{attribute 'linkalways'} 
{attribute 'no_explicit_call' := 'This FB is a CLASS and must be accessed using methods or properties'}
{attribute 'enable_dynamic_creation'}
FUNCTION_BLOCK FINAL GT_SINT EXTENDS Node
VAR
	in1 : _SINT(0);
	in2 : _SINT(0);
	out : _BOOL(FALSE);
END_VAR

METHOD PUBLIC Clone : I_Node
VAR
	pNode : POINTER TO GT_SINT;
END_VAR
pNode := __NEW(GT_SINT);
Clone := pNode^;
END_METHOD

METHOD FB_init : BOOL
VAR_INPUT
	bInitRetains : BOOL; // if TRUE, the retain variables are initialized (warm start / cold start)
	bInCopyCode : BOOL;  // if TRUE, the instance afterwards gets moved into the copy code (online change)
END_VAR
AddInput('in1',THIS^.in1);
AddInput('in2',THIS^.in2);
AddOutput('out', THIS^.out);
END_METHOD

METHOD PROTECTED OnExecute
VAR
END_VAR
out.Value := in1.Value > in2.Value;
END_METHOD

END_FUNCTION_BLOCK

(* stored: Version 1.1.0.1, ProductVersion 3.1.4024.15
   POU GT_SINT: Id {69151acb-79db-46e5-8e03-585d68b75999}, SpecialFunc None
   Folder Constructor: Id {1a6696ee-6d7e-4616-8718-6fcead4db9f0}
   Method Clone: Id {fcc5539b-ce54-410d-a691-fd40c100d57f}
   Method FB_init: Id {1cfb7cab-c464-4778-a61d-cb2eb5cd5385}
   Method OnExecute: Id {0155bf89-6e10-4d8c-b93f-fab1a91bdd5e} *)
